// Interlock logic for the Carbide Shutter
FUNCTION F_CarbideShutterEnable : BOOL
VAR_INPUT
	bMasterOverride : BOOL; //Master manual override control input
END_VAR
VAR_IN_OUT CONSTANT
	stErrors : ST_ErrorStates; // Currently detected errors
END_VAR
VAR
END_VAR

IF (stErrors.bHardwareFailure // Close carbide shutter if there is a hardware failure
	OR stErrors.bLeakOpcpaCarbideOn (* OR stErrors.bLeakUnderTable *) ) // Close carbide shutter if leak in OPCPA with carbide on or if there is a leak under the table
	AND NOT bMasterOverride //if master override is TRUE, ignore all errors
THEN
	F_CarbideShutterEnable := FALSE;
ELSE
	F_CarbideShutterEnable := TRUE;
END_IF

END_FUNCTION

(* stored: Version 1.1.0.1, ProductVersion 3.1.4024.6
   POU F_CarbideShutterEnable: Id {9a18bc5e-2ef3-4837-9298-88db836b21d8}, SpecialFunc None *)
